// LS Electric XG5000 project: 9-2
// PLC LSPLC

PROGRAM NewProgram (task: 스캔 프로그램)

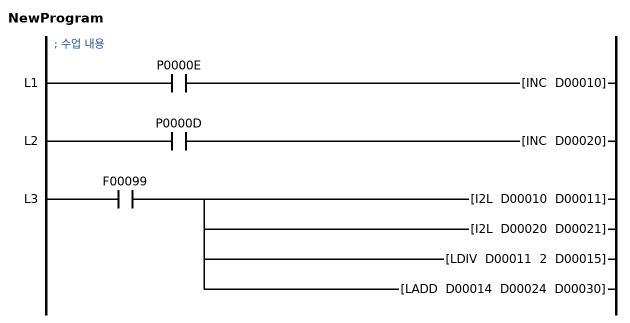
// 수업 내용
; L1
LOAD      P0000E
INC       D00010
; L2
LOAD      P0000D
INC       D00020
; L3
LOAD      F00099
I2L       D00010 D00011
I2L       D00020 D00021
LDIV      D00011 2 D00015
LADD      D00014 D00024 D00030